// Mitsubishi GX Works2 project: PULSE   PLC: Q03UDV

PROGRAM MAIN
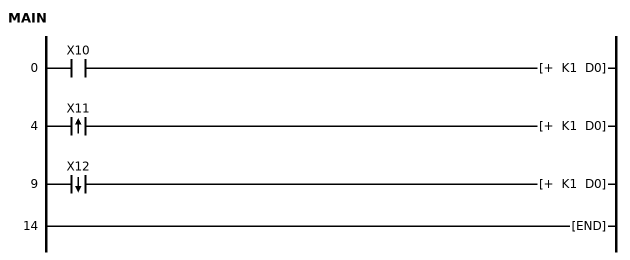
0     LD      X10
      +       K1 D0
4     LDP     X11
      +       K1 D0
9     LDF     X12
      +       K1 D0
14    END
END_PROGRAM
